	W =   -36.298 deg,	P =   -14.510 deg,	R =   128.300 deg
   GP2:
	UF : 1, UT : 1,
	J1=    80.000 deg,	J2=    90.000 deg
};
P[1001]{
   GP1:
	UF : 1, UT : 1,		CONFIG : 'N U T, 0, 0, 0',
	X =  2511.729  mm,	Y =  -421.925  mm,	Z =   -58.540  mm,
	W =   -23.404 deg,	P =   -31.780 deg,	R =    95.153 deg
   GP2:
	UF : 1, UT : 1,
	J1=    80.000 deg,	J2=    90.000 deg
};
P[1002]{
   GP1:
	UF : 1, UT : 1,		CONFIG : 'N U T, 0, 0, 0',
	X =  2535.771  mm,	Y =  -433.252  mm,	Z =   -64.743  mm,
	W =   -18.432 deg,	P =   -37.731 deg,	R =   100.748 deg
   GP2:
	UF : 1, UT : 1,
	J1=    80.000 deg,	J2=    90.000 deg
};
P[1003]{
   GP1:
	UF : 1, UT : 1,		CONFIG : 'N U T, 0, 0, 0',
	X =  2556.962  mm,	Y =  -440.220  mm,	Z =   -66.569  mm,
	W =   -18.755 deg,	P =   -39.987 deg,	R =   104.532 deg
   GP2:
	UF : 1, UT : 1,
	J1=    80.000 deg,	J2=    90.000 deg
};
P[1004]{
   GP1:
	UF : 1, UT : 1,		CONFIG : 'N U T, 0, 0, 0',
	X =  2567.777  mm,	Y =  -444.328  mm,	Z =   -68.493  mm,
	W =   -18.759 deg,	P =   -39.992 deg,	R =   104.538 deg
   GP2:
	UF : 1, UT : 1,
	J1=    80.000 deg,	J2=    90.000 deg
};
P[1005]{
   GP1:
	UF : 1, UT : 1,		CONFIG : 'N U T, 0, 0, 0',
	X =  2613.677  mm,	Y =  -477.273  mm,	Z =   -77.598  mm,
	W =   -35.261 deg,	P =   -23.936 deg,	R =   103.297 deg
   GP2:
	UF : 1, UT : 1,
	J1=    80.000 deg,	J2=    90.000 deg
};
P[1006]{
   GP1:
	UF : 1, UT : 1,		CONFIG : 'N U T, 0, 0, 0',
	X =  2626.463  mm,	Y =  -510.442  mm,	Z =   -79.962  mm,
	W =   -33.013 deg,	P =   -16.162 deg,	R =    67.004 deg
   GP2:
	UF : 1, UT : 1,
	J1=    80.000 deg,	J2=    90.000 deg
};
P[1007]{
   GP1:
	UF : 1, UT : 1,		CONFIG : 'N U T, 0, 0, 0',
	X =  2625.741  mm,	Y =  -708.057  mm,	Z =   -78.550  mm,
	W =   -27.676 deg,	P =   -22.323 deg,	R =    54.093 deg
   GP2:
	UF : 1, UT : 1,
	J1=    80.000 deg,	J2=    90.000 deg
};
P[1008]{
   GP1:
	UF : 1, UT : 1,		CONFIG : 'N U T, 0, 0, 0',
	X =  2553.477  mm,	Y =  -818.838  mm,	Z =   -68.643  mm,
	W =   -27.687 deg,	P =   -22.317 deg,	R =    54.099 deg
   GP2:
	UF : 1, UT : 1,
	J1=    80.000 deg,	J2=    90.000 deg
};
P[1009]{
   GP1:
	UF : 1, UT : 1,		CONFIG : 'N U T, 0, 0, 0',
	X =  2554.187  mm,	Y =  -807.503  mm,	Z =   -67.688  mm,
	W =   -27.687 deg,	P =   -22.318 deg,	R =    54.099 deg
   GP2:
	UF : 1, UT : 1,
	J1=    80.000 deg,	J2=    90.000 deg
};
P[1010]{
   GP1:
	UF : 1, UT : 1,		CONFIG : 'N U T, 0, 0, 0',
	X =  2563.526  mm,	Y =  -794.948  mm,	Z =   -70.177  mm,
	W =   -27.684 deg,	P =   -22.320 deg,	R =    23.347 deg
   GP2:
	UF : 1, UT : 1,
	J1=    80.000 deg,	J2=    90.000 deg
};
P[1011]{
   GP1:
	UF : 1, UT : 1,		CONFIG : 'N U T, 0, 0, 0',
	X =  2575.827  mm,	Y =  -789.432  mm,	Z =   -72.319  mm,
	W =   -33.338 deg,	P =   -11.310 deg,	R =    17.619 deg
   GP2:
	UF : 1, UT : 1,
	J1=    80.000 deg,	J2=    90.000 deg
};
P[1012]{
   GP1:
	UF : 1, UT : 1,		CONFIG : 'N U T, 0, 0, 0',
	X =  2614.220  mm,	Y =  -761.078  mm,	Z =   -80.341  mm,
	W =   -30.065 deg,	P =    -4.703 deg,	R =    42.983 deg
   GP2:
	UF : 1, UT : 1,
	J1=    80.000 deg,	J2=    90.000 deg
};
P[1013]{
   GP1:
	UF : 1, UT : 1,		CONFIG : 'N U T, 0, 0, 0',
	X =  2630.670  mm,	Y =  -703.014  mm,	Z =   -79.942  mm,
	W =   -25.583 deg,	P =   -24.734 deg,	R =    48.847 deg
   GP2:
	UF : 1, UT : 1,
	J1=    80.000 deg,	J2=    90.000 deg
};
P[1014]{
   GP1:
	UF : 1, UT : 1,		CONFIG : 'N U T, 0, 0, -1',
	X =  2500.101  mm,	Y =  -843.989  mm,	Z =      .763  mm,
	W =   -44.579 deg,	P =    -6.906 deg,	R =    84.731 deg
   GP2:
	UF : 1, UT : 1,
	J1=    90.000 deg,	J2=   -90.000 deg
};
P[1015]{
   GP1:
	UF : 1, UT : 1,		CONFIG : 'N U T, 0, 0, -1',
	X =  2498.506  mm,	Y =  -772.585  mm,	Z =      .733  mm,
	W =   -44.581 deg,	P =    -6.907 deg,	R =    84.733 deg
   GP2:
	UF : 1, UT : 1,
	J1=    90.000 deg,	J2=   -90.000 deg
};
P[1016]{
   GP1:
	UF : 1, UT : 1,		CONFIG : 'N U T, 0, 0, 0',
	X =  2525.148  mm,	Y =  -742.055  mm,	Z =     1.319  mm,
	W =   -39.980 deg,	P =    14.825 deg,	R =    17.711 deg
   GP2:
	UF : 1, UT : 1,
	J1=    90.000 deg,	J2=   -90.000 deg
};
P[1017]{
   GP1:
	UF : 1, UT : 1,		CONFIG : 'N U T, 0, 0, 0',
	X =  2567.357  mm,	Y =  -744.379  mm,	Z =    -1.238  mm,
	W =   -39.977 deg,	P =    14.826 deg,	R =    17.707 deg
   GP2:
	UF : 1, UT : 1,
	J1=    90.000 deg,	J2=   -90.000 deg
};
P[1018]{
   GP1:
	UF : 1, UT : 1,		CONFIG : 'N U T, 0, 0, 0',
	X =  2754.219  mm,	Y =  -152.494  mm,	Z =   181.656  mm,
	W =    -1.647 deg,	P =    -7.141 deg,	R =    13.038 deg
   GP2:
	UF : 1, UT : 1,
	J1=    90.000 deg,	J2=  -135.000 deg
};
P[1019]{
   GP1:
	UF : 1, UT : 1,		CONFIG : 'N U T, 0, 0, 0',
	X =  2871.009  mm,	Y =  -153.833  mm,	Z =   186.035  mm,
	W =    -5.452 deg,	P =   -22.504 deg,	R =    14.011 deg
   GP2:
	UF : 1, UT : 1,
	J1=    90.000 deg,	J2=  -135.000 deg
};
P[1020]{
   GP1:
	UF : 1, UT : 1,		CONFIG : 'N U T, 0, 0, 0',
	X =  2382.307  mm,	Y =  -257.240  mm,	Z =    90.661  mm,
	W =     -.006 deg,	P =      .007 deg,	R =    -2.933 deg
   GP2:
	UF : 1, UT : 1,
	J1=    90.000 deg,	J2=  -135.000 deg
};
P[1021]{
   GP1:
	UF : 1, UT : 1,		CONFIG : 'N U T, 0, 0, 0',
	X =  2759.554  mm,	Y =  -256.153  mm,	Z =    93.128  mm,
	W =      .075 deg,	P =    -1.490 deg,	R =    -2.941 deg
   GP2:
	UF : 1, UT : 1,
	J1=    90.000 deg,	J2=  -135.000 deg
};
P[1022]{
   GP1:
	UF : 1, UT : 1,		CONFIG : 'N U T, 0, 0, 0',
	X =  2509.947  mm,	Y =   181.457  mm,	Z =    -1.616  mm,
	W =    37.876 deg,	P =   -26.378 deg,	R =    31.551 deg
   GP2:
	UF : 1, UT : 1,
	J1=    90.000 deg,	J2=   -90.000 deg
};
P[1023]{
   GP1:
	UF : 1, UT : 1,		CONFIG : 'N U T, 0, 0, 0',
	X =  2462.907  mm,	Y =   180.747  mm,	Z =    -1.513  mm,
	W =    37.870 deg,	P =   -26.389 deg,	R =    31.565 deg
   GP2:
	UF : 1, UT : 1,
	J1=    90.000 deg,	J2=   -90.000 deg
};
P[1024]{
   GP1:
	UF : 1, UT : 1,		CONFIG : 'N U T, 0, 0, 0',
	X =  2445.326  mm,	Y =   180.108  mm,	Z =      .250  mm,
	W =    40.547 deg,	P =   -21.447 deg,	R =    53.219 deg
   GP2:
	UF : 1, UT : 1,
	J1=    90.000 deg,	J2=   -90.000 deg
};
P[1025]{
   GP1:
	UF : 1, UT : 1,		CONFIG : 'N U T, 0, 0, 0',
	X =  1690.038  mm,	Y =   -49.964  mm,	Z =   -11.982  mm,
	W =    41.392 deg,	P =    19.516 deg,	R =   -17.038 deg
   GP2:
	UF : 1, UT : 1,
	J1=    90.000 deg,	J2=   -90.000 deg
};
P[1026]{
   GP1:
	UF : 1, UT : 1,		CONFIG : 'N U T, 0, 0, 0',
	X =  1652.969  mm,	Y =   -49.284  mm,	Z =   -12.616  mm,
	W =    41.393 deg,	P =    19.516 deg,	R =   -16.113 deg
   GP2:
	UF : 1, UT : 1,
	J1=    90.000 deg,	J2=   -90.000 deg
};
P[1027]{
   GP1:
	UF : 1, UT : 1,		CONFIG : 'N U T, 0, 0, 0',
	X =  1642.910  mm,	Y =   -50.885  mm,	Z =   -11.965  mm,
	W =    41.394 deg,	P =    19.515 deg,	R =     3.468 deg
   GP2:
	UF : 1, UT : 1,
	J1=    90.000 deg,	J2=   -90.000 deg
};
P[1028]{
   GP1:
	UF : 1, UT : 1,		CONFIG : 'N U T, 0, 0, 0',
	X =  1634.473  mm,	Y =   -53.135  mm,	Z =   -14.299  mm,
	W =    41.393 deg,	P =    19.522 deg,	R =    24.098 deg
   GP2:
	UF : 1, UT : 1,
	J1=    90.000 deg,	J2=   -90.000 deg
};
P[1029]{
   GP1:
	UF : 1, UT : 1,		CONFIG : 'N U T, 0, 0, 0',
	X =  1608.240  mm,	Y =   -80.496  mm,	Z =   -13.783  mm,
	W =    37.029 deg,	P =    27.662 deg,	R =    15.297 deg
   GP2:
	UF : 1, UT : 1,
	J1=    90.000 deg,	J2=   -90.000 deg
};
P[1030]{
   GP1:
	UF : 1, UT : 1,		CONFIG : 'N U T, 0, 0, 0',
	X =  1588.769  mm,	Y =   -91.533  mm,	Z =   -13.038  mm,
	W =    38.934 deg,	P =    23.606 deg,	R =   -29.718 deg
   GP2:
	UF : 1, UT : 1,
	J1=    90.000 deg,	J2=   -90.000 deg
};
P[1031]{
   GP1:
	UF : 1, UT : 1,		CONFIG : 'N U T, 0, 0, 0',
	X =  1569.200  mm,	Y =   -66.418  mm,	Z =   -14.762  mm,
	W =    36.734 deg,	P =    28.084 deg,	R =  -109.083 deg
   GP2:
	UF : 1, UT : 1,
	J1=    90.000 deg,	J2=   -90.000 deg
};
P[1032]{
   GP1:
	UF : 1, UT : 1,		CONFIG : 'N U T, 0, 0, 0',
	X =  1565.612  mm,	Y =   -24.282  mm,	Z =   -16.223  mm,
	W =    36.733 deg,	P =    28.086 deg,	R =  -114.514 deg
   GP2:
	UF : 1, UT : 1,
	J1=    90.000 deg,	J2=   -90.000 deg
};
P[1033]{
   GP1:
	UF : 1, UT : 1,		CONFIG : 'N U T, 0, 0, 0',
	X =  1562.317  mm,	Y =   -16.001  mm,	Z =   -12.611  mm,
	W =    36.725 deg,	P =    28.084 deg,	R =   -80.637 deg
   GP2:
	UF : 1, UT : 1,
	J1=    90.000 deg,	J2=   -90.000 deg
};
P[1034]{
   GP1:
	UF : 1, UT : 1,		CONFIG : 'N U T, 0, 0, 0',
	X =  1553.848  mm,	Y =   -10.188  mm,	Z =   -12.900  mm,
	W =    36.731 deg,	P =    28.089 deg,	R =   -43.974 deg
   GP2:
	UF : 1, UT : 1,
	J1=    90.000 deg,	J2=   -90.000 deg
};
P[1035]{
   GP1:
	UF : 1, UT : 1,		CONFIG : 'N U T, 0, 0, 0',
	X =  1547.336  mm,	Y =    -8.620  mm,	Z =   -13.271  mm,
	W =    36.729 deg,	P =    28.089 deg,	R =   -43.983 deg
   GP2:
	UF : 1, UT : 1,
	J1=    90.000 deg,	J2=   -90.000 deg
};
P[1036]{
   GP1:
	UF : 1, UT : 1,		CONFIG : 'N U T, 0, 0, 0',
	X =  2367.321  mm,	Y =   184.102  mm,	Z =    -3.691  mm,
	W =    38.118 deg,	P =   -25.963 deg,	R =    27.293 deg
   GP2:
	UF : 1, UT : 1,
	J1=    90.000 deg,	J2=   -90.000 deg
};
P[1037]{
   GP1:
	UF : 1, UT : 1,		CONFIG : 'N U T, 0, 0, 0',
	X =  2406.160  mm,	Y =   183.060  mm,	Z =    -3.000  mm,
	W =    38.129 deg,	P =   -25.958 deg,	R =    27.290 deg
   GP2:
	UF : 1, UT : 1,
	J1=    90.000 deg,	J2=   -90.000 deg
};
P[1038]{
   GP1:
	UF : 1, UT : 1,		CONFIG : 'N U T, 0, 0, 0',
	X =  2428.050  mm,	Y =   179.285  mm,	Z =     1.204  mm,
	W =    11.741 deg,	P =   -38.464 deg,	R =    42.116 deg
   GP2:
	UF : 1, UT : 1,
	J1=    89.989 deg,	J2=   -90.001 deg
};
P[1039]{
   GP1:
	UF : 1, UT : 1,		CONFIG : 'N U T, 0, 0, 0',
	X =  1668.666  mm,	Y =   205.664  mm,	Z =   -12.534  mm,
	W =   -36.933 deg,	P =    22.769 deg,	R =   -15.981 deg
   GP2:
	UF : 1, UT : 1,
	J1=    90.000 deg,	J2=   -90.000 deg
};
P[1040]{
   GP1:
	UF : 1, UT : 1,		CONFIG : 'N U T, 0, 0, 0',
	X =  1703.657  mm,	Y =   203.883  mm,	Z =   -12.893  mm,
	W =   -36.939 deg,	P =    22.781 deg,	R =    39.328 deg
   GP2:
	UF : 1, UT : 1,
	J1=    90.000 deg,	J2=   -90.000 deg
};
P[1041]{
   GP1:
	UF : 1, UT : 1,		CONFIG : 'N U T, 0, 0, 0',
	X =  1979.129  mm,	Y =   205.388  mm,	Z =   -13.477  mm,
	W =   -36.938 deg,	P =    22.781 deg,	R =    39.327 deg
   GP2:
	UF : 1, UT : 1,
	J1=    90.000 deg,	J2=   -90.000 deg
};
P[1042]{
   GP1:
	UF : 1, UT : 1,		CONFIG : 'N U T, 0, 0, 0',
	X =  1995.822  mm,	Y =   203.251  mm,	Z =   -10.207  mm,
	W =   -40.748 deg,	P =    13.395 deg,	R =    62.817 deg
   GP2:
	UF : 1, UT : 1,
	J1=    90.000 deg,	J2=   -90.000 deg
};
P[1043]{
   GP1:
	UF : 1, UT : 1,		CONFIG : 'N U T, 0, 0, 0',
	X =  2395.612  mm,	Y =    98.485  mm,	Z =   -19.732  mm,
	W =   -47.023 deg,	P =     6.661 deg,	R =   -51.409 deg
   GP2:
	UF : 1, UT : 1,
	J1=    83.000 deg,	J2=   -90.000 deg
};
P[1044]{
   GP1:
	UF : 1, UT : 1,		CONFIG : 'N U T, 0, 0, 0',
	X =  2391.596  mm,	Y =   124.389  mm,	Z =   -21.745  mm,
	W =   -46.999 deg,	P =     6.652 deg,	R =   -83.994 deg
   GP2:
	UF : 1, UT : 1,
	J1=    83.000 deg,	J2=   -90.000 deg
};
P[1045]{
   GP1:
	UF : 1, UT : 1,		CONFIG : 'N U T, 0, 0, 0',
	X =  2392.331  mm,	Y =   158.473  mm,	Z =   -19.448  mm,
	W =   -47.981 deg,	P =     7.880 deg,	R =   -87.080 deg
   GP2:
	UF : 1, UT : 1,
	J1=    83.000 deg,	J2=   -90.000 deg
};
P[1046]{
   GP1:
	UF : 1, UT : 1,		CONFIG : 'N U T, 0, 0, 0',
	X =  2391.390  mm,	Y =   184.030  mm,	Z =   -21.542  mm,
	W =   -51.565 deg,	P =    20.299 deg,	R =  -107.020 deg
   GP2:
	UF : 1, UT : 1,
	J1=    83.000 deg,	J2=   -90.000 deg
};
P[1047]{
   GP1:
	UF : 1, UT : 1,		CONFIG : 'N U T, 0, 0, 0',
	X =  2366.000  mm,	Y =   195.031  mm,	Z =    -5.475  mm,
	W =   -44.811 deg,	P =    -4.561 deg,	R =    -2.490 deg
   GP2:
	UF : 1, UT : 1,
	J1=    90.000 deg,	J2=   -90.000 deg
};
P[1048]{
   GP1:
	UF : 1, UT : 1,		CONFIG : 'N U T, 0, 0, 0',
	X =  2509.255  mm,	Y =   194.275  mm,	Z =    -4.194  mm,
	W =   -44.809 deg,	P =    -4.555 deg,	R =    -2.481 deg
   GP2:
	UF : 1, UT : 1,
	J1=    90.000 deg,	J2=   -90.000 deg
};
P[1049]{
   GP1:
	UF : 1, UT : 1,		CONFIG : 'N U T, 0, 0, 0',
	X =  2367.908  mm,	Y =    96.138  mm,	Z =    -4.435  mm,
	W =   -44.397 deg,	P =     8.168 deg,	R =    14.048 deg
   GP2:
	UF : 1, UT : 1,
	J1=    90.000 deg,	J2=   -90.000 deg
};
P[1050]{
   GP1:
	UF : 1, UT : 1,		CONFIG : 'N U T, 0, 0, 0',
	X =  2413.075  mm,	Y =    96.166  mm,	Z =    -3.839  mm,
	W =   -44.394 deg,	P =     8.166 deg,	R =    14.048 deg
   GP2:
	UF : 1, UT : 1,
	J1=    90.000 deg,	J2=   -90.000 deg
};
P[1051]{
   GP1:
	UF : 1, UT : 1,		CONFIG : 'N U T, 0, 0, 0',
	X =  2427.383  mm,	Y =    97.382  mm,	Z =     -.048  mm,
	W =   -44.529 deg,	P =    -7.125 deg,	R =    33.229 deg
   GP2:
	UF : 1, UT : 1,
	J1=    90.000 deg,	J2=   -90.000 deg
};
P[1052]{
   GP1:
	UF : 1, UT : 1,		CONFIG : 'N U T, 0, 0, 0',
	X =  2337.427  mm,	Y =    71.440  mm,	Z =   847.749  mm,
	W =    45.399 deg,	P =    17.266 deg,	R =    -1.541 deg
   GP2:
	UF : 1, UT : 1,
	J1=    90.000 deg,	J2=   -90.000 deg
};
P[1053]{
   GP1:
	UF : 1, UT : 1,		CONFIG : 'N U T, 0, 0, 0',
	X =  2402.831  mm,	Y =   104.785  mm,	Z =   847.602  mm,
	W =    45.390 deg,	P =    17.268 deg,	R =    -1.529 deg
   GP2:
	UF : 1, UT : 1,
	J1=    90.000 deg,	J2=   -90.000 deg
};
P[1054]{
   GP1:
	UF : 1, UT : 1,		CONFIG : 'N U T, 0, 0, 0',
	X =  2402.842  mm,	Y =   109.949  mm,	Z =   847.942  mm,
	W =     1.452 deg,	P =    40.371 deg,	R =    26.792 deg
   GP2:
	UF : 1, UT : 1,
	J1=    90.000 deg,	J2=   -90.000 deg
};
P[1055]{
   GP1:
	UF : 1, UT : 1,		CONFIG : 'N U T, 0, 0, 0',
	X =  2392.403  mm,	Y =   126.094  mm,	Z =   845.932  mm,
	W =     1.448 deg,	P =    40.368 deg,	R =    26.765 deg
   GP2:
	UF : 1, UT : 1,
	J1=    90.000 deg,	J2=   -90.000 deg
};
P[1056]{
   GP1:
	UF : 1, UT : 1,		CONFIG : 'F U T, 0, 0, 0',
	X =  2325.472  mm,	Y =    92.116  mm,	Z =   847.036  mm,
	W =   -46.230 deg,	P =   -25.147 deg,	R =    34.050 deg
   GP2:
	UF : 1, UT : 1,
	J1=    90.000 deg,	J2=   -90.000 deg
};
P[1057]{
   GP1:
	UF : 1, UT : 1,		CONFIG : 'F U T, 0, 0, 0',
	X =  2391.645  mm,	Y =   126.896  mm,	Z =   847.777  mm,
	W =   -46.222 deg,	P =   -25.150 deg,	R =    34.042 deg
   GP2:
	UF : 1, UT : 1,
	J1=    90.000 deg,	J2=   -90.000 deg
};
P[1058]{
   GP1:
	UF : 1, UT : 1,		CONFIG : 'N U T, 0, 0, 0',
	X =  2011.750  mm,	Y =   -80.950  mm,	Z =    -4.575  mm,
	W =    40.372 deg,	P =    23.935 deg,	R =    74.339 deg
   GP2:
	UF : 1, UT : 1,
	J1=    90.000 deg,	J2=  -100.000 deg
};
P[1059]{
   GP1:
	UF : 1, UT : 1,		CONFIG : 'N U T, 0, 0, 0',
	X =  2007.194  mm,	Y =   142.177  mm,	Z =   -45.001  mm,
	W =    45.685 deg,	P =     4.509 deg,	R =    78.826 deg
   GP2:
	UF : 1, UT : 1,
	J1=    90.000 deg,	J2=  -100.000 deg
};
P[1060]{
   GP1:
	UF : 1, UT : 1,		CONFIG : 'N U T, 0, 0, 0',
	X =  2229.070  mm,	Y =   -48.871  mm,	Z =     4.516  mm,
	W =    44.904 deg,	P =    -3.411 deg,	R =     3.413 deg
   GP2:
	UF : 1, UT : 1,
	J1=    90.000 deg,	J2=   -90.000 deg
};
P[1061]{
   GP1:
	UF : 1, UT : 1,		CONFIG : 'N U T, 0, 0, 0',
	X =  2266.341  mm,	Y =   -46.762  mm,	Z =     3.253  mm,
	W =    44.893 deg,	P =    -3.421 deg,	R =     3.427 deg
   GP2:
	UF : 1, UT : 1,
	J1=    90.000 deg,	J2=   -90.000 deg
};
P[1062]{
   GP1:
	UF : 1, UT : 1,		CONFIG : 'N U T, 0, 0, 0',
	X =  2142.334  mm,	Y =   -48.860  mm,	Z =    -3.830  mm,
	W =    44.883 deg,	P =     3.632 deg,	R =    -4.928 deg
   GP2:
	UF : 1, UT : 1,
	J1=    90.000 deg,	J2=   -90.000 deg
};
P[1063]{
   GP1:
	UF : 1, UT : 1,		CONFIG : 'N U T, 0, 0, 0',
	X =  2212.734  mm,	Y =   -47.597  mm,	Z =    -4.519  mm,
	W =    44.886 deg,	P =     3.634 deg,	R =    -4.918 deg
   GP2:
	UF : 1, UT : 1,
	J1=    90.000 deg,	J2=   -90.000 deg
};
P[1064]{
   GP1:
	UF : 1, UT : 1,		CONFIG : 'N U T, 0, 0, 0',
	X =  2216.176  mm,	Y =   -46.694  mm,	Z =    -5.378  mm,
	W =    44.882 deg,	P =     3.630 deg,	R =   -11.556 deg
   GP2:
	UF : 1, UT : 1,
	J1=    90.000 deg,	J2=   -90.000 deg
};
P[1065]{
   GP1:
	UF : 1, UT : 1,		CONFIG : 'N U T, 0, 0, 0',
	X =  1992.932  mm,	Y =   -47.776  mm,	Z =   -14.567  mm,
	W =    44.891 deg,	P =     3.636 deg,	R =    -8.860 deg
   GP2:
	UF : 1, UT : 1,
	J1=    90.000 deg,	J2=   -90.000 deg
};
P[1066]{
   GP1:
	UF : 1, UT : 1,		CONFIG : 'N U T, 0, 0, 0',
	X =  2106.099  mm,	Y =   -46.333  mm,	Z =   -15.544  mm,
	W =    44.875 deg,	P =     3.623 deg,	R =    -8.839 deg
   GP2:
	UF : 1, UT : 1,
	J1=    90.000 deg,	J2=   -90.000 deg
};
P[1067]{
   GP1:
	UF : 1, UT : 1,		CONFIG : 'N U T, 0, 0, 0',
	X =  2117.103  mm,	Y =   -50.973  mm,	Z =   -11.238  mm,
	W =    41.211 deg,	P =   -19.950 deg,	R =    -8.037 deg
   GP2:
	UF : 1, UT : 1,
	J1=    90.000 deg,	J2=   -90.000 deg
};
P[1068]{
   GP1:
	UF : 1, UT : 1,		CONFIG : 'N U T, 0, 0, 0',
	X =  2075.732  mm,	Y =  -109.868  mm,	Z =   -15.932  mm,
	W =   -37.504 deg,	P =      .971 deg,	R =    76.657 deg
   GP2:
	UF : 1, UT : 1,
	J1=    90.000 deg,	J2=   -90.000 deg
};
P[1069]{
   GP1:
	UF : 1, UT : 1,		CONFIG : 'N U T, 0, 0, 0',
	X =  2112.001  mm,	Y =   -75.797  mm,	Z =   -17.252  mm,
	W =   -37.498 deg,	P =      .974 deg,	R =    85.226 deg
   GP2:
	UF : 1, UT : 1,
	J1=    90.000 deg,	J2=   -90.000 deg
};
P[1070]{
   GP1:
	UF : 1, UT : 1,		CONFIG : 'N U T, 0, 0, 0',
	X =  2126.497  mm,	Y =   -60.152  mm,	Z =   -12.916  mm,
	W =   -48.237 deg,	P =     4.570 deg,	R =   105.632 deg
   GP2:
	UF : 1, UT : 1,
	J1=    89.995 deg,	J2=   -90.001 deg
};
P[1071]{
   GP1:
	UF : 1, UT : 1,		CONFIG : 'N U T, 0, 0, 1',
	X =  2137.360  mm,	Y =  -144.268  mm,	Z =   834.187  mm,
	W =      .668 deg,	P =    41.811 deg,	R =  -160.738 deg
   GP2:
	UF : 1, UT : 1,
	J1=    90.000 deg,	J2=   -90.000 deg
};
P[1072]{
   GP1:
	UF : 1, UT : 1,		CONFIG : 'N U T, 0, 0, 1',
	X =  2144.152  mm,	Y =  -167.358  mm,	Z =   834.668  mm,
	W =      .532 deg,	P =    40.619 deg,	R =  -160.815 deg
   GP2:
	UF : 1, UT : 1,
	J1=    90.000 deg,	J2=   -90.000 deg
};
P[1073]{
   GP1:
	UF : 1, UT : 1,		CONFIG : 'N U T, 0, 0, 0',
	X =  2131.457  mm,	Y =  -193.376  mm,	Z =   832.812  mm,
	W =    -1.789 deg,	P =    43.352 deg,	R =   109.759 deg
   GP2:
	UF : 1, UT : 1,
	J1=    90.000 deg,	J2=   -90.000 deg
};
P[1074]{
   GP1:
	UF : 1, UT : 1,		CONFIG : 'N U T, 0, 0, 0',
	X =  2099.029  mm,	Y =  -181.626  mm,	Z =   831.918  mm,
	W =      .955 deg,	P =    43.489 deg,	R =    21.015 deg
   GP2:
	UF : 1, UT : 1,
	J1=    90.000 deg,	J2=   -90.000 deg
};
P[1075]{
   GP1:
	UF : 1, UT : 1,		CONFIG : 'N U T, 0, 0, 0',
	X =  2085.167  mm,	Y =  -135.110  mm,	Z =   833.287  mm,
	W =      .566 deg,	P =    42.530 deg,	R =    14.578 deg
   GP2:
	UF : 1, UT : 1,
	J1=    90.000 deg,	J2=   -90.000 deg
};
P[1076]{
   GP1:
	UF : 1, UT : 1,		CONFIG : 'N U T, 0, 0, 0',
	X =  2104.005  mm,	Y =  -110.952  mm,	Z =   833.109  mm,
	W =      .858 deg,	P =    43.011 deg,	R =   -74.577 deg
   GP2:
	UF : 1, UT : 1,
	J1=    90.000 deg,	J2=   -90.000 deg
};
P[1077]{
   GP1:
	UF : 1, UT : 1,		CONFIG : 'N U T, 0, 0, 0',
	X =  2131.832  mm,	Y =  -123.512  mm,	Z =   834.193  mm,
	W =      .102 deg,	P =    42.115 deg,	R =  -162.102 deg
   GP2:
	UF : 1, UT : 1,
	J1=    90.000 deg,	J2=   -90.000 deg
};
P[1078]{
   GP1:
	UF : 1, UT : 1,		CONFIG : 'N U T, 0, 0, 0',
	X =  2138.893  mm,	Y =  -144.672  mm,	Z =   833.681  mm,
	W =      .505 deg,	P =    42.850 deg,	R =  -163.809 deg
   GP2:
	UF : 1, UT : 1,
	J1=    90.000 deg,	J2=   -90.000 deg
};
P[1079]{
   GP1:
	UF : 1, UT : 1,		CONFIG : 'N U T, 0, 0, 0',
	X =  2107.700  mm,	Y =  -213.626  mm,	Z =   831.846  mm,
	W =     -.446 deg,	P =    39.556 deg,	R =   -90.694 deg
   GP2:
	UF : 1, UT : 1,
	J1=    90.000 deg,	J2=   -90.000 deg
};
P[1080]{
   GP1:
	UF : 1, UT : 1,		CONFIG : 'N U T, 0, 0, 0',
	X =  2200.131  mm,	Y =  -214.897  mm,	Z =   833.980  mm,
	W =     -.446 deg,	P =    39.557 deg,	R =   -90.713 deg
   GP2:
	UF : 1, UT : 1,
	J1=    90.000 deg,	J2=   -90.000 deg
};
P[1081]{
   GP1:
	UF : 1, UT : 1,		CONFIG : 'N U T, 0, 0, 0',
	X =  2212.289  mm,	Y =  -210.992  mm,	Z =   834.347  mm,
	W =     -.442 deg,	P =    39.558 deg,	R =   -57.815 deg
   GP2:
	UF : 1, UT : 1,
	J1=    90.000 deg,	J2=   -90.000 deg
};
P[1082]{
   GP1:
	UF : 1, UT : 1,		CONFIG : 'N U T, 0, 0, 0',
	X =  2220.486  mm,	Y =  -200.207  mm,	Z =   832.598  mm,
	W =     -.448 deg,	P =    39.556 deg,	R =   -44.056 deg
   GP2:
	UF : 1, UT : 1,
	J1=    90.000 deg,	J2=   -90.000 deg
};
P[1083]{
   GP1:
	UF : 1, UT : 1,		CONFIG : 'N U T, 0, 0, 0',
	X =  2441.776  mm,	Y =    55.830  mm,	Z =   833.792  mm,
	W =      .117 deg,	P =    42.766 deg,	R =   -42.899 deg
   GP2:
	UF : 1, UT : 1,
	J1=    90.000 deg,	J2=   -90.000 deg
};
P[1084]{
   GP1:
	UF : 1, UT : 1,		CONFIG : 'N U T, 0, 0, 0',
	X =  2448.836  mm,	Y =    63.315  mm,	Z =   833.149  mm,
	W =      .109 deg,	P =    42.766 deg,	R =   -49.058 deg
   GP2:
	UF : 1, UT : 1,
	J1=    90.000 deg,	J2=   -90.000 deg
};
P[1085]{
   GP1:
	UF : 1, UT : 1,		CONFIG : 'N U T, 0, 0, 0',
	X =  2455.189  mm,	Y =    65.446  mm,	Z =   835.378  mm,
	W =      .109 deg,	P =    42.768 deg,	R =   -56.123 deg
   GP2:
	UF : 1, UT : 1,
	J1=    90.000 deg,	J2=   -90.000 deg
};
P[1086]{
   GP1:
	UF : 1, UT : 1,		CONFIG : 'N U T, 0, 0, 0',
	X =  2645.172  mm,	Y =   206.772  mm,	Z =   838.084  mm,
	W =    29.497 deg,	P =    29.459 deg,	R =    -6.841 deg
   GP2:
	UF : 1, UT : 1,
	J1=    90.000 deg,	J2=   -90.000 deg
};
P[1087]{
   GP1:
	UF : 1, UT : 1,		CONFIG : 'N U T, 0, 0, 0',
	X =  2652.713  mm,	Y =   210.527  mm,	Z =   838.644  mm,
	W =    29.493 deg,	P =    29.463 deg,	R =    -6.844 deg
   GP2:
	UF : 1, UT : 1,
	J1=    90.000 deg,	J2=   -90.000 deg
};
P[1088]{
   GP1:
	UF : 1, UT : 1,		CONFIG : 'N U T, 0, 0, 0',
	X =  1967.929  mm,	Y =   -36.946  mm,	Z =    54.617  mm,
	W =   -51.899 deg,	P =     9.369 deg,	R =    14.299 deg
   GP2:
	UF : 1, UT : 1,
	J1=    90.000 deg,	J2=   -90.000 deg
};
P[1089]{
   GP1:
	UF : 1, UT : 1,		CONFIG : 'N U T, 0, 0, 0',
	X =  1952.806  mm,	Y =   -38.944  mm,	Z =    52.063  mm,
	W =   -51.882 deg,	P =     9.361 deg,	R =     5.846 deg
   GP2:
	UF : 1, UT : 1,
	J1=    90.000 deg,	J2=   -90.000 deg
};
P[1090]{
   GP1:
	UF : 1, UT : 1,		CONFIG : 'N U T, 0, 0, 0',
	X =  1695.004  mm,	Y =   -37.169  mm,	Z =    53.060  mm,
	W =   -51.893 deg,	P =     9.370 deg,	R =     5.849 deg
   GP2:
	UF : 1, UT : 1,
	J1=    90.000 deg,	J2=   -90.000 deg
};
P[1091]{
   GP1:
	UF : 1, UT : 1,		CONFIG : 'N U T, 0, 0, 0',
	X =  1671.652  mm,	Y =   -33.229  mm,	Z =    53.086  mm,
	W =   -51.882 deg,	P =     9.363 deg,	R =   -32.598 deg
   GP2:
	UF : 1, UT : 1,
	J1=    90.000 deg,	J2=   -90.000 deg
};
P[1092]{
   GP1:
	UF : 1, UT : 1,		CONFIG : 'N U T, 0, 0, 0',
	X =  2229.154  mm,	Y =   -35.668  mm,	Z =      .956  mm,
	W =   -45.065 deg,	P =    -5.945 deg,	R =    -3.251 deg
   GP2:
	UF : 1, UT : 1,
	J1=    90.000 deg,	J2=   -90.000 deg
};
P[1093]{
   GP1:
	UF : 1, UT : 1,		CONFIG : 'N U T, 0, 0, 0',
	X =  2263.854  mm,	Y =   -39.114  mm,	Z =    -2.230  mm,
	W =   -45.063 deg,	P =    -5.945 deg,	R =    -3.254 deg
   GP2:
	UF : 1, UT : 1,
	J1=    90.000 deg,	J2=   -90.000 deg
};
P[1094]{
   GP1:
	UF : 1, UT : 1,		CONFIG : 'N U T, 0, 0, 0',
	X =  2143.762  mm,	Y =   -38.233  mm,	Z =    -9.450  mm,
	W =   -46.267 deg,	P =    -5.650 deg,	R =    -4.455 deg
   GP2:
	UF : 1, UT : 1,
	J1=    89.999 deg,	J2=   -90.000 deg
};
P[1095]{
   GP1:
	UF : 1, UT : 1,		CONFIG : 'N U T, 0, 0, 0',
	X =  2211.456  mm,	Y =   -38.697  mm,	Z =   -10.423  mm,
	W =   -44.729 deg,	P =    -5.487 deg,	R =    -5.519 deg
   GP2:
	UF : 1, UT : 1,
	J1=    90.000 deg,	J2=   -90.000 deg
};
P[1096]{
   GP1:
	UF : 1, UT : 1,		CONFIG : 'N U T, 0, 0, 0',
	X =  2213.501  mm,	Y =   -38.329  mm,	Z =    -9.533  mm,
	W =   -44.727 deg,	P =    -5.491 deg,	R =    10.507 deg
   GP2:
	UF : 1, UT : 1,
	J1=    90.000 deg,	J2=   -90.000 deg
};
P[1097]{
   GP1:
	UF : 1, UT : 1,		CONFIG : 'N U T, 0, 0, 0',
	X =  2115.187  mm,	Y =   -36.549  mm,	Z =   -16.802  mm,
	W =   -44.729 deg,	P =    -5.491 deg,	R =    -5.515 deg
   GP2:
	UF : 1, UT : 1,
	J1=    90.000 deg,	J2=   -90.000 deg
};
P[1098]{
   GP1:
	UF : 1, UT : 1,		CONFIG : 'N U T, 0, 0, 0',
	X =  2031.075  mm,	Y =   -35.591  mm,	Z =   -15.945  mm,
	W =   -44.726 deg,	P =    -5.493 deg,	R =    -5.522 deg
   GP2:
	UF : 1, UT : 1,
	J1=    90.000 deg,	J2=   -90.000 deg
};
P[1099]{
   GP1:
	UF : 1, UT : 1,		CONFIG : 'N U T, 0, 0, 0',
	X =  2012.774  mm,	Y =   -33.603  mm,	Z =   -16.255  mm,
	W =   -44.728 deg,	P =    -5.488 deg,	R =   -41.543 deg
   GP2:
	UF : 1, UT : 1,
	J1=    90.000 deg,	J2=   -90.000 deg
};
P[1100]{
   GP1:
	UF : 1, UT : 1,		CONFIG : 'N U T, 0, 0, 0',
	X =  1659.349  mm,	Y =   229.576  mm,	Z =   -15.827  mm,
	W =    34.860 deg,	P =    26.474 deg,	R =  -126.851 deg
   GP2:
	UF : 1, UT : 1,
	J1=    90.000 deg,	J2=   -90.000 deg
};
P[1101]{
   GP1:
	UF : 1, UT : 1,		CONFIG : 'N U T, 0, 0, 1',
	X =  1662.403  mm,	Y =    10.748  mm,	Z =   -16.240  mm,
	W =    36.966 deg,	P =    27.691 deg,	R =  -122.597 deg
   GP2:
	UF : 1, UT : 1,
	J1=    90.000 deg,	J2=   -90.000 deg
};
P[1102]{
   GP1:
	UF : 1, UT : 1,		CONFIG : 'N U T, 0, 0, 0',
	X =  1661.230  mm,	Y =   -12.152  mm,	Z =   -15.927  mm,
	W =    37.079 deg,	P =    27.798 deg,	R =  -137.823 deg
   GP2:
	UF : 1, UT : 1,
	J1=    90.000 deg,	J2=   -90.000 deg
};
P[1103]{
   GP1:
	UF : 1, UT : 1,		CONFIG : 'N U T, 0, 0, 0',
	X =  2070.256  mm,	Y =   -29.016  mm,	Z =    17.551  mm,
	W =    27.122 deg,	P =    24.041 deg,	R =  -162.981 deg
   GP2:
	UF : 1, UT : 1,
	J1=    80.000 deg,	J2=   -90.000 deg
};
P[1104]{
   GP1:
	UF : 1, UT : 1,		CONFIG : 'N U T, 0, 0, 1',
	X =  2077.472  mm,	Y =     9.268  mm,	Z =    15.852  mm,
	W =    26.540 deg,	P =    23.907 deg,	R =  -139.393 deg
   GP2:
	UF : 1, UT : 1,
	J1=    80.000 deg,	J2=   -90.000 deg
};
P[1105]{
   GP1:
	UF : 1, UT : 1,		CONFIG : 'N U T, 0, 0, 0',
	X =  2079.821  mm,	Y =    18.267  mm,	Z =    15.557  mm,
	W =    26.544 deg,	P =    23.915 deg,	R =  -163.856 deg
   GP2:
	UF : 1, UT : 1,
	J1=    80.000 deg,	J2=   -90.000 deg
};
P[1106]{
   GP1:
	UF : 1, UT : 1,		CONFIG : 'N U T, 0, 0, 0',
	X =  2088.621  mm,	Y =    27.690  mm,	Z =    13.857  mm,
	W =    17.944 deg,	P =    33.024 deg,	R =   153.337 deg
   GP2:
	UF : 1, UT : 1,
	J1=    80.000 deg,	J2=   -90.000 deg
};
P[1107]{
   GP1:
	UF : 1, UT : 1,		CONFIG : 'N U T, 0, 0, 0',
	X =  2236.640  mm,	Y =   176.401  mm,	Z =    -7.067  mm,
	W =     2.794 deg,	P =    36.171 deg,	R =   129.508 deg
   GP2:
	UF : 1, UT : 1,
	J1=    80.000 deg,	J2=   -90.000 deg
};
P[1108]{
   GP1:
	UF : 1, UT : 1,		CONFIG : 'N U T, 0, 0, 0',
	X =  2264.963  mm,	Y =   203.116  mm,	Z =   -13.114  mm,
	W =     3.306 deg,	P =    33.869 deg,	R =   124.421 deg
   GP2:
	UF : 1, UT : 1,
	J1=    80.000 deg,	J2=   -90.000 deg
};
P[1109]{
   GP1:
	UF : 1, UT : 1,		CONFIG : 'N U T, 0, 0, 0',
	X =  2287.031  mm,	Y =   217.729  mm,	Z =   -16.695  mm,
	W =     6.006 deg,	P =    35.930 deg,	R =   123.381 deg
   GP2:
	UF : 1, UT : 1,
	J1=    80.000 deg,	J2=   -90.000 deg
};
P[1110]{
   GP1:
	UF : 1, UT : 1,		CONFIG : 'N U T, 0, 0, 0',
	X =  2387.696  mm,	Y =   277.952  mm,	Z =   -35.568  mm,
	W =     8.794 deg,	P =    37.204 deg,	R =   129.070 deg
   GP2:
	UF : 1, UT : 1,
	J1=    80.000 deg,	J2=   -90.000 deg
};
P[1111]{
   GP1:
	UF : 1, UT : 1,		CONFIG : 'N U T, 0, 0, 0',
	X =  2404.670  mm,	Y =   288.506  mm,	Z =   -40.636  mm,
	W =    -2.498 deg,	P =    34.190 deg,	R =   123.664 deg
   GP2:
	UF : 1, UT : 1,
	J1=    80.000 deg,	J2=   -90.000 deg
};
P[1112]{
   GP1:
	UF : 1, UT : 1,		CONFIG : 'N U T, 0, 0, 0',
	X =  2423.597  mm,	Y =   314.103  mm,	Z =   -39.372  mm,
	W =      .578 deg,	P =    31.082 deg,	R =   135.853 deg
   GP2:
	UF : 1, UT : 1,
	J1=    80.000 deg,	J2=   -90.000 deg
};
P[1113]{
   GP1:
	UF : 1, UT : 1,		CONFIG : 'N U T, 0, 0, 0',
	X =  2506.157  mm,	Y =   429.784  mm,	Z =   -53.556  mm,
	W =   -18.684 deg,	P =    29.858 deg,	R =   100.231 deg
   GP2:
	UF : 1, UT : 1,
	J1=    80.000 deg,	J2=   -90.000 deg
};
P[1114]{
   GP1:
	UF : 1, UT : 1,		CONFIG : 'N U T, 0, 0, 0',
	X =  2522.874  mm,	Y =   447.428  mm,	Z =   -56.211  mm,
	W =   -18.818 deg,	P =    32.562 deg,	R =    79.861 deg
   GP2:
	UF : 1, UT : 1,
	J1=    80.000 deg,	J2=   -90.000 deg
};
P[1115]{
   GP1:
	UF : 1, UT : 1,		CONFIG : 'N U T, 0, 0, 0',
	X =  2554.598  mm,	Y =   458.467  mm,	Z =   -62.590  mm,
	W =   -16.507 deg,	P =    33.838 deg,	R =    74.968 deg
   GP2:
	UF : 1, UT : 1,
	J1=    80.000 deg,	J2=   -90.000 deg
};
P[1116]{
   GP1:
	UF : 1, UT : 1,		CONFIG : 'N U T, 0, 0, 0',
	X =  2567.108  mm,	Y =   460.127  mm,	Z =   -64.835  mm,
	W =   -16.506 deg,	P =    33.836 deg,	R =    74.958 deg
   GP2:
	UF : 1, UT : 1,
	J1=    80.000 deg,	J2=   -90.000 deg
};
P[1117]{
   GP1:
	UF : 1, UT : 1,		CONFIG : 'N U T, 0, 0, 0',
	X =  2609.688  mm,	Y =   486.425  mm,	Z =   -71.766  mm,
	W =   -17.685 deg,	P =    33.469 deg,	R =   110.387 deg
   GP2:
	UF : 1, UT : 1,
	J1=    80.000 deg,	J2=   -90.000 deg
};
P[1118]{
   GP1:
	UF : 1, UT : 1,		CONFIG : 'N U T, 0, 0, 0',
	X =  2628.545  mm,	Y =   536.100  mm,	Z =   -75.597  mm,
	W =   -28.178 deg,	P =    11.271 deg,	R =   110.042 deg
   GP2:
	UF : 1, UT : 1,
	J1=    80.000 deg,	J2=   -90.000 deg
};
P[1119]{
   GP1:
	UF : 1, UT : 1,		CONFIG : 'N U T, 0, 0, 0',
	X =  2632.222  mm,	Y =   732.009  mm,	Z =   -80.623  mm,
	W =   -28.919 deg,	P =    12.962 deg,	R =   109.016 deg
   GP2:
	UF : 1, UT : 1,
	J1=    80.000 deg,	J2=   -90.000 deg
};
P[1120]{
   GP1:
	UF : 1, UT : 1,		CONFIG : 'N U T, 0, 0, 0',
	X =  2634.037  mm,	Y =   736.946  mm,	Z =   -80.036  mm,
	W =   -28.912 deg,	P =    12.964 deg,	R =    86.663 deg
   GP2:
	UF : 1, UT : 1,
	J1=    80.000 deg,	J2=   -90.000 deg
};
P[1121]{
   GP1:
	UF : 1, UT : 1,		CONFIG : 'N U T, 0, 0, 0',
	X =  2636.521  mm,	Y =   741.783  mm,	Z =   -80.114  mm,
	W =   -28.912 deg,	P =    12.964 deg,	R =    81.290 deg
   GP2:
	UF : 1, UT : 1,
	J1=    80.000 deg,	J2=   -90.000 deg
};
P[1122]{
   GP1:
	UF : 1, UT : 1,		CONFIG : 'N U T, 0, 0, 0',
	X =  2643.067  mm,	Y =   762.281  mm,	Z =   -80.422  mm,
	W =   -29.832 deg,	P =     9.276 deg,	R =    88.856 deg
   GP2:
	UF : 1, UT : 1,
	J1=    80.000 deg,	J2=   -90.000 deg
};
P[1123]{
   GP1:
	UF : 1, UT : 1,		CONFIG : 'N U T, 0, 0, 0',
	X =  2640.869  mm,	Y =   777.391  mm,	Z =   -80.196  mm,
	W =   -33.768 deg,	P =      .740 deg,	R =   112.866 deg
   GP2:
	UF : 1, UT : 1,
	J1=    80.000 deg,	J2=   -90.000 deg
};
P[1124]{
   GP1:
	UF : 1, UT : 1,		CONFIG : 'N U T, 0, 0, 0',
	X =  2554.805  mm,	Y =   840.968  mm,	Z =   -65.386  mm,
	W =   -31.195 deg,	P =     9.618 deg,	R =   105.424 deg
   GP2:
	UF : 1, UT : 1,
	J1=    80.000 deg,	J2=   -90.000 deg
};
P[1125]{
   GP1:
	UF : 1, UT : 1,		CONFIG : 'N U T, 0, 0, 0',
	X =  2556.195  mm,	Y =   827.922  mm,	Z =   -66.293  mm,
	W =   -32.481 deg,	P =     1.245 deg,	R =    91.949 deg
   GP2:
	UF : 1, UT : 1,
	J1=    80.000 deg,	J2=   -90.000 deg
};
P[1126]{
   GP1:
	UF : 1, UT : 1,		CONFIG : 'N U T, 0, 0, 0',
	X =  2562.628  mm,	Y =   816.135  mm,	Z =   -66.477  mm,
	W =   -29.304 deg,	P =   -14.723 deg,	R =   104.306 deg
   GP2:
	UF : 1, UT : 1,
	J1=    80.000 deg,	J2=   -90.000 deg
};
P[1127]{
   GP1:
	UF : 1, UT : 1,		CONFIG : 'N U T, 0, 0, 0',
	X =  2576.087  mm,	Y =   812.043  mm,	Z =   -72.164  mm,
	W =    -3.300 deg,	P =   -34.456 deg,	R =   105.021 deg
   GP2:
	UF : 1, UT : 1,
	J1=    80.000 deg,	J2=   -90.000 deg
};
P[1128]{
   GP1:
	UF : 1, UT : 1,		CONFIG : 'N U T, 0, 0, 0',
	X =  2599.271  mm,	Y =   811.663  mm,	Z =   -77.249  mm,
	W =    -3.299 deg,	P =   -34.461 deg,	R =   105.020 deg
   GP2:
	UF : 1, UT : 1,
	J1=    80.000 deg,	J2=   -90.000 deg
};
P[1129]{
   GP1:
	UF : 1, UT : 1,		CONFIG : 'N U T, 0, 0, 0',
	X =  2617.323  mm,	Y =   805.644  mm,	Z =   -77.465  mm,
	W =     3.038 deg,	P =   -34.483 deg,	R =    65.938 deg
   GP2:
	UF : 1, UT : 1,
	J1=    80.000 deg,	J2=   -90.000 deg
};
P[1130]{
   GP1:
	UF : 1, UT : 1,		CONFIG : 'N U T, 0, 0, 0',
	X =  2640.391  mm,	Y =   775.794  mm,	Z =   -80.773  mm,
	W =   -11.649 deg,	P =   -32.807 deg,	R =    38.714 deg
   GP2:
	UF : 1, UT : 1,
	J1=    80.000 deg,	J2=   -90.000 deg
};
P[1131]{
   GP1:
	UF : 1, UT : 1,		CONFIG : 'N U T, 0, 0, 0',
	X =  1063.279  mm,	Y = -1053.306  mm,	Z =   783.332  mm,
	W =    24.557 deg,	P =   -38.977 deg,	R =    -6.176 deg
   GP2:
	UF : 1, UT : 1,
	J1=   180.000 deg,	J2=  -150.000 deg
};
P[1132]{
   GP1:
	UF : 1, UT : 1,		CONFIG : 'N U T, 0, 0, 0',
	X =  1109.166  mm,	Y = -1127.961  mm,	Z =   780.009  mm,
	W =    24.527 deg,	P =   -38.988 deg,	R =    -6.133 deg
   GP2:
	UF : 1, UT : 1,
	J1=   180.000 deg,	J2=  -150.000 deg
};
P[1133]{
   GP1:
	UF : 1, UT : 1,		CONFIG : 'N U T, 0, 0, 0',
	X =   786.252  mm,	Y =  -573.217  mm,	Z =   780.478  mm,
	W =   -27.530 deg,	P =    35.491 deg,	R =   168.461 deg
   GP2:
	UF : 1, UT : 1,
	J1=   180.000 deg,	J2=  -150.000 deg
};
P[1134]{
   GP1:
	UF : 1, UT : 1,		CONFIG : 'N U T, 0, 0, 0',
	X =   927.792  mm,	Y =  -818.010  mm,	Z =   778.982  mm,
	W =   -27.603 deg,	P =    35.465 deg,	R =   163.373 deg
   GP2:
	UF : 1, UT : 1,
	J1=   180.000 deg,	J2=  -150.000 deg
};
P[1135]{
   GP1:
	UF : 1, UT : 1,		CONFIG : 'N U T, 0, 0, 0',
	X =  1047.239  mm,	Y = -1021.242  mm,	Z =   783.994  mm,
	W =    33.109 deg,	P =    30.260 deg,	R =  -102.113 deg
   GP2:
	UF : 1, UT : 1,
	J1=   180.000 deg,	J2=  -150.000 deg
};
P[1136]{
   GP1:
	UF : 1, UT : 1,		CONFIG : 'N U T, 0, 0, 0',
	X =   765.614  mm,	Y =  -535.452  mm,	Z =   786.067  mm,
	W =    41.849 deg,	P =   -18.077 deg,	R =   -40.922 deg
   GP2:
	UF : 1, UT : 1,
	J1=   180.000 deg,	J2=  -150.000 deg
};
P[1137]{
   GP1:
	UF : 1, UT : 1,		CONFIG : 'N U T, 0, 0, 0',
	X =   721.837  mm,	Y =  -462.053  mm,	Z =   783.548  mm,
	W =    27.769 deg,	P =   -36.841 deg,	R =   -11.320 deg
   GP2:
	UF : 1, UT : 1,
	J1=   180.000 deg,	J2=  -150.000 deg
};
P[1138]{
   GP1:
	UF : 1, UT : 1,		CONFIG : 'N U T, 0, 0, 0',
	X =  1898.693  mm,	Y = -1465.196  mm,	Z =  1035.174  mm,
	W =   -39.886 deg,	P =    23.861 deg,	R =    23.910 deg
   GP2:
	UF : 1, UT : 1,
	J1=   180.000 deg,	J2=   -90.000 deg
};
P[1139]{
   GP1:
	UF : 1, UT : 1,		CONFIG : 'N U T, 0, 0, 0',
	X =  1930.842  mm,	Y = -1465.932  mm,	Z =  1036.894  mm,
	W =   -43.540 deg,	P =    14.560 deg,	R =    14.833 deg
   GP2:
	UF : 1, UT : 1,
	J1=   180.000 deg,	J2=   -90.000 deg
};
P[1140]{
   GP1:
	UF : 1, UT : 1,		CONFIG : 'N U T, 0, 0, 0',
	X =  1966.391  mm,	Y = -1464.791  mm,	Z =  1037.270  mm,
	W =   -43.537 deg,	P =    14.558 deg,	R =    14.821 deg
   GP2:
	UF : 1, UT : 1,
	J1=   180.000 deg,	J2=   -90.000 deg
};
P[1141]{
   GP1:
	UF : 1, UT : 1,		CONFIG : 'N U T, 0, 0, 0',
	X =  1996.744  mm,	Y = -1479.610  mm,	Z =  1035.370  mm,
	W =   -43.544 deg,	P =    14.560 deg,	R =   -14.022 deg
   GP2:
	UF : 1, UT : 1,
	J1=   180.000 deg,	J2=   -90.000 deg
};
P[1142]{
   GP1:
	UF : 1, UT : 1,		CONFIG : 'N U T, 0, 0, 0',
	X =  2005.341  mm,	Y = -1493.994  mm,	Z =  1032.872  mm,
	W =   -44.808 deg,	P =     8.522 deg,	R =   -27.704 deg
   GP2:
	UF : 1, UT : 1,
	J1=   180.000 deg,	J2=   -90.000 deg
};
P[1143]{
   GP1:
	UF : 1, UT : 1,		CONFIG : 'N U T, 0, 0, 0',
	X =  1897.818  mm,	Y =  1491.288  mm,	Z =  1034.377  mm,
	W =    41.278 deg,	P =    19.806 deg,	R =   -17.231 deg
   GP2:
	UF : 1, UT : 1,
	J1=   180.000 deg,	J2=    90.000 deg
};
P[1144]{
   GP1:
	UF : 1, UT : 1,		CONFIG : 'N U T, 0, 0, 0',
	X =  1932.829  mm,	Y =  1488.728  mm,	Z =  1037.568  mm,
	W =    41.270 deg,	P =    19.801 deg,	R =   -17.222 deg
   GP2:
	UF : 1, UT : 1,
	J1=   180.000 deg,	J2=    90.000 deg
};
P[1145]{
   GP1:
	UF : 1, UT : 1,		CONFIG : 'N U T, 0, 0, 0',
	X =  1964.476  mm,	Y =  1486.706  mm,	Z =  1040.490  mm,
	W =    41.276 deg,	P =    19.802 deg,	R =   -17.225 deg
   GP2:
	UF : 1, UT : 1,
	J1=   180.000 deg,	J2=    90.000 deg
};
P[1146]{
   GP1:
	UF : 1, UT : 1,		CONFIG : 'N U T, 0, 0, 0',
	X =  1987.397  mm,	Y =  1501.086  mm,	Z =  1037.179  mm,
	W =    41.274 deg,	P =    19.802 deg,	R =     6.738 deg
   GP2:
	UF : 1, UT : 1,
	J1=   180.000 deg,	J2=    90.000 deg
};
P[1147]{
   GP1:
	UF : 1, UT : 1,		CONFIG : 'N U T, 0, 0, 0',
	X =  1995.872  mm,	Y =  1510.585  mm,	Z =  1037.723  mm,
	W =    43.860 deg,	P =    11.269 deg,	R =    16.934 deg
   GP2:
	UF : 1, UT : 1,
	J1=   180.000 deg,	J2=    90.000 deg
};
P[1148]{
   GP1:
	UF : 1, UT : 1,		CONFIG : 'N U T, 0, 0, 0',
	X =  1652.192  mm,	Y = -1411.641  mm,	Z =  1037.125  mm,
	W =   -42.857 deg,	P =   -15.295 deg,	R =    39.125 deg
   GP2:
	UF : 1, UT : 1,
	J1=   180.000 deg,	J2=  -125.000 deg
};
P[1149]{
   GP1:
	UF : 1, UT : 1,		CONFIG : 'N U T, 0, 0, 0',
	X =  1657.327  mm,	Y = -1402.491  mm,	Z =  1038.261  mm,
	W =   -42.570 deg,	P =   -16.799 deg,	R =    40.477 deg
   GP2:
	UF : 1, UT : 1,
	J1=   180.000 deg,	J2=  -125.000 deg
};
P[1150]{
   GP1:
	UF : 1, UT : 1,		CONFIG : 'N U T, 0, 0, 0',
	X =  1673.592  mm,	Y = -1391.668  mm,	Z =  1036.866  mm,
	W =   -42.572 deg,	P =   -16.799 deg,	R =    43.540 deg
   GP2:
	UF : 1, UT : 1,
	J1=   180.000 deg,	J2=  -125.000 deg
};
P[1151]{
   GP1:
	UF : 1, UT : 1,		CONFIG : 'N U T, 0, 0, 0',
	X =  1678.567  mm,	Y = -1386.491  mm,	Z =  1039.737  mm,
	W =   -43.819 deg,	P =   -18.072 deg,	R =    47.125 deg
   GP2:
	UF : 1, UT : 1,
	J1=   180.000 deg,	J2=  -125.000 deg
};
P[1152]{
   GP1:
	UF : 1, UT : 1,		CONFIG : 'F U T, 0, 0, 0',
	X =  1107.454  mm,	Y =  1017.315  mm,	Z =  1037.603  mm,
	W =    44.131 deg,	P =    -6.201 deg,	R =   -51.550 deg
   GP2:
	UF : 1, UT : 1,
	J1=   180.000 deg,	J2=   150.000 deg
};
P[1153]{
   GP1:
	UF : 1, UT : 1,		CONFIG : 'F U T, 0, 0, 0',
	X =  1116.811  mm,	Y =  1013.553  mm,	Z =  1037.422  mm,
	W =    43.027 deg,	P =    -7.259 deg,	R =   -34.946 deg
   GP2:
	UF : 1, UT : 1,
	J1=   180.000 deg,	J2=   150.000 deg
};
P[1154]{
   GP1:
	UF : 1, UT : 1,		CONFIG : 'F U T, 0, 0, 0',
	X =  1131.215  mm,	Y =  1008.607  mm,	Z =  1040.074  mm,
	W =    42.657 deg,	P =   -14.123 deg,	R =   -20.713 deg
   GP2:
	UF : 1, UT : 1,
	J1=   180.000 deg,	J2=   150.000 deg
};
P[1155]{
   GP1:
	UF : 1, UT : 1,		CONFIG : 'F U T, 0, 0, 0',
	X =  1138.823  mm,	Y =  1009.249  mm,	Z =  1040.961  mm,
	W =    42.642 deg,	P =   -14.134 deg,	R =   -27.083 deg
   GP2:
	UF : 1, UT : 1,
	J1=   180.000 deg,	J2=   150.000 deg
};
P[1162]{
   GP1:
	UF : 1, UT : 1,		CONFIG : 'N U T, 0, 0, 0',
	X =  2793.017  mm,	Y = -1472.744  mm,	Z =   939.115  mm,
	W =   -37.776 deg,	P =   -31.389 deg,	R =    42.831 deg
   GP2:
	UF : 1, UT : 1,
	J1=   100.000 deg,	J2=   -90.000 deg
};
P[1163]{
   GP1:
	UF : 1, UT : 1,		CONFIG : 'N U T, 0, 0, 0',
	X =  2794.995  mm,	Y = -1494.504  mm,	Z =   937.599  mm,
	W =   -37.762 deg,	P =   -31.393 deg,	R =    42.829 deg
   GP2:
	UF : 1, UT : 1,
	J1=   100.000 deg,	J2=   -90.000 deg
};
P[1164]{
   GP1:
	UF : 1, UT : 1,		CONFIG : 'N U T, 0, 0, 0',
	X =  2786.501  mm,	Y = -1525.976  mm,	Z =   936.000  mm,
	W =   -42.869 deg,	P =   -22.972 deg,	R =    39.989 deg
   GP2:
	UF : 1, UT : 1,
	J1=    99.999 deg,	J2=   -90.000 deg
};
P[1165]{
   GP1:
	UF : 1, UT : 1,		CONFIG : 'N U T, 0, 0, 0',
	X =  2776.812  mm,	Y = -1537.743  mm,	Z =   933.598  mm,
	W =   -45.701 deg,	P =   -14.897 deg,	R =    35.260 deg
   GP2:
	UF : 1, UT : 1,
	J1=   100.000 deg,	J2=   -90.000 deg
};
P[1166]{
   GP1:
	UF : 1, UT : 1,		CONFIG : 'N U T, 0, 0, 0',
	X =  2742.053  mm,	Y = -1559.698  mm,	Z =   926.134  mm,
	W =   -45.722 deg,	P =   -14.879 deg,	R =    30.415 deg
   GP2:
	UF : 1, UT : 1,
	J1=   100.000 deg,	J2=   -90.000 deg
};
P[1167]{
   GP1:
	UF : 1, UT : 1,		CONFIG : 'N U T, 0, 0, 0',
	X =  2723.925  mm,	Y = -1565.150  mm,	Z =   922.276  mm,
	W =   -45.707 deg,	P =   -14.888 deg,	R =    18.304 deg
   GP2:
	UF : 1, UT : 1,
	J1=   100.000 deg,	J2=   -90.000 deg
};
P[1168]{
   GP1:
	UF : 1, UT : 1,		CONFIG : 'N U T, 0, 0, 0',
	X =  2711.316  mm,	Y = -1566.584  mm,	Z =   918.265  mm,
	W =   -45.711 deg,	P =   -14.879 deg,	R =     6.076 deg
   GP2:
	UF : 1, UT : 1,
	J1=   100.000 deg,	J2=   -90.000 deg
};
P[1169]{
   GP1:
	UF : 1, UT : 1,		CONFIG : 'N U T, 0, 0, 0',
	X =  2683.065  mm,	Y = -1567.564  mm,	Z =   912.242  mm,
	W =   -45.718 deg,	P =   -14.888 deg,	R =     6.082 deg
   GP2:
	UF : 1, UT : 1,
	J1=   100.000 deg,	J2=   -90.000 deg
};
/END
